(* PLC project CoDeSys External Library Template, WAGO e!COCKPIT e!COCKPIT, author 3S - Smart Software Solutions GmbH *)
(* stored: creationDateTime 2019-10-29T12:22:40.4802773, version 3.5.5.30, modificationDateTime 2019-10-24T14:40:07.960949, organization 3S - Smart Software Solutions GmbH *)
(* Library project template with all possible element types, docu and a sample project structure *)

(* values of enumPPPSWezelClimatixPOL63xError: BrakKomunikacji: brak komunikacji z zadajnikiem; AlarmOgolnyBezpieczenstwa: alarm ogólny bezpieczeństwa; AlarmOgolnyKrytyczny: alarm ogólny krytyczny; AlarmOgolnyOstrzezenie: alarm ogólny ostrzeżenie; AlarmOgolnyInformacyjny: alarm ogólny informacyjny; AlarmCzujnikaZewnetrznego: alarm braku zmiany wartości czujnika temp. zewnetrznj; AlarmCzujnikaZasilaniaObwoduHC1: alarm braku zmiany wartości czujnika temp. zasilana obwodu HC1; AlarmCzujnikaZasilaniaObwoduDHW: alarm braku zmiany wartości czujnika temp. zasilana obwodu DHW; AlarmBrakuOsiagnieciaTemperaturyHC1: alarm braku osiągnięcia temp. zadanej obwodu HC1; AlarmBrakuOsiagnieciaTemperaturyDHW: alarm braku osiągnięcia temp. zadanej obwodu DHW; BladIloscPomiarowTemperatury: alarm zbyt małej ilości pomiarów dokonanych w ciągu dnia do obliczenia średniej *)

(* Autor: Paweł Kąkol, 2018-09-03-PK Prawa majątkowe: Solwena Sp. z o.o., Aktualizacje: 2019-02-14-AWy: dodanie alarmów czujników temp. zewnętrznej i zasilania obwodu HC1, DHW Opis: enum służy do obsługi alarmów w fb węzła Climatix POL63x na budynkach PPP Sopot (ENGIE) *)
{attribute 'qualified_only'}
{attribute 'strict'}
TYPE enumPPPSWezelClimatixPOL63xError : (BrakKomunikacji := 1, AlarmOgolnyBezpieczenstwa := 2, AlarmOgolnyKrytyczny := 3, AlarmOgolnyOstrzezenie := 4, AlarmOgolnyInformacyjny := 5, AlarmCzujnikaZewnetrznego := 6, AlarmCzujnikaZasilaniaObwoduHC1 := 7, AlarmCzujnikaZasilaniaObwoduDHW := 8, AlarmBrakuOsiagnieciaTemperaturyHC1 := 9, AlarmBrakuOsiagnieciaTemperaturyDHW := 10, BladIloscPomiarowTemperatury := 11);
END_TYPE
